FUNCTION_BLOCK FB_StateReadParameters IMPLEMENTS I_State
VAR
	_refMainStateMachine		: REFERENCE TO FB_MainStateMachine;
	_fbXmlSrvRead				: FB_XmlSrvRead;
	_fbTcAlarm					: FB_TcAlarm;
END_VAR

METHOD GetDescription : STRING
GetDescription := 'Read parameters';
END_METHOD

METHOD ClearErrors
_fbTcAlarm.Clear(
	nTimeStamp			:= 0,
	bResetConfirmation	:= TRUE);
END_METHOD

METHOD StopButtonPressed
END_METHOD

METHOD StartButtonPressed
END_METHOD

METHOD Execute
_fbXmlSrvRead(
	pSymAddr	:= ADR(MachineParameters.stData),
	cbSymSize	:= SIZEOF(MachineParameters.stData),
	sFilePath	:= MachineParameters.sFilePath,
	sXPath		:= MachineParameters.sXPath,
	bExecute	:= TRUE);

IF NOT _fbXmlSrvRead.bBusy AND NOT _fbXmlSrvRead.bError THEN
	_fbXmlSrvRead(bExecute := FALSE);
	_refMainStateMachine.SetState(_refMainStateMachine.ipStateEStop);
ELSIF NOT _fbXmlSrvRead.bBusy AND _fbXmlSrvRead.bError THEN
	_fbTcAlarm.ipArguments.Clear().AddUDInt(_fbXmlSrvRead.nErrId);
	_fbTcAlarm.Raise(0);
	_fbXmlSrvRead(bExecute := FALSE);
	_refMainStateMachine.SetState(_refMainStateMachine.ipStateError);
END_IF
END_METHOD

METHOD FB_init : BOOL
VAR_INPUT
	// if TRUE, the retain variables are initialized (warm start / cold start)
	bInitRetains			: BOOL;
	// if TRUE, the instance afterwards gets moved into the copy code (online
	// change)
	bInCopyCode				: BOOL;
	fbMainStateMachine		: REFERENCE TO FB_MainStateMachine;
END_VAR
_refMainStateMachine REF= fbMainStateMachine;
_fbTcAlarm.CreateEx(
	stEventEntry		:= TC_EVENTS.StatePatternEvents.ParameterReadError,
	bWithConfirmation	:= FALSE,
	ipSourceInfo		:= 0);
END_METHOD

METHOD SafetyTripped
END_METHOD

METHOD SafetyAcknowledged
END_METHOD

END_FUNCTION_BLOCK

(* stored: Version 1.1.0.1, ProductVersion 3.1.4024.11
   POU FB_StateReadParameters: Id {d06eba43-4d67-4414-9ab9-44be67d2f02c}, SpecialFunc None
   Method GetDescription: Id {2858806e-5883-4242-bc9a-02865edc683d}
   Method ClearErrors: Id {2e17538e-57b6-4db0-8ea4-cbda233cbdc3}
   Method StopButtonPressed: Id {445be649-727c-4203-8d2d-78693d8e3145}
   Method StartButtonPressed: Id {5a10994b-3f3f-4e40-b6a6-e4b0aab8e025}
   Method Execute: Id {7469fe26-825a-4e09-92c5-86ca59062f26}
   Method FB_init: Id {a3f9f64f-c1df-4d42-b14e-58c4ec93f78f}
   Method SafetyTripped: Id {a4e20ab1-79a2-4599-b9a0-5c8799b4ac89}
   Method SafetyAcknowledged: Id {f9dac850-8892-44ec-98c1-cffca2efbe6e} *)
